{attribute 'linkalways'} 
{attribute 'no_explicit_call' := 'This FB is a CLASS and must be accessed using methods or properties'}
{attribute 'enable_dynamic_creation'}
FUNCTION_BLOCK Node_F_VN_AppendToContainer_ITcVnContainer EXTENDS VisionNode
VAR
    ipElement : _ITcVnContainer;
    ipContainer : _ITcVnContainer;
    hrPrev : _HRESULT(S_OK);
	hresult : _HRESULT(S_OK);
END_VAR

METHOD PUBLIC  Clone : I_Node
VAR
	pNode : POINTER TO Node_F_VN_AppendToContainer_ITcVnContainer;
END_VAR
pNode := __NEW(Node_F_VN_AppendToContainer_ITcVnContainer);
Clone := pNode^;
END_METHOD

METHOD FB_init : BOOL
VAR_INPUT
	bInitRetains : BOOL; // if TRUE, the retain variables are initialized (warm start / cold start)
	bInCopyCode : BOOL;  // if TRUE, the instance afterwards gets moved into the copy code (online change)
END_VAR
AddInput('ipElement', ipElement);
AddInput('ipContainer', ipContainer);
AddInput('hrPrev', hrPrev);
AddOutput('ipContainer', ipContainer);
AddOutput('hresult',hresult);
END_METHOD

METHOD PROTECTED OnExecute : HRESULT
hresult.Value := F_VN_AppendToContainer_ITcVnContainer(
    ipElement := ipElement.Value,
	ipContainer := ipContainer.Value,
	hrPrev:= hrPrev.Value);
END_METHOD

METHOD PUBLIC PreExecutionCheck
VAR_INPUT
	Check : I_PreExecutionChecks;
END_VAR
Check.IsTrue(ipContainer.IsValid, 'ipContainer must be a valid container');
END_METHOD

END_FUNCTION_BLOCK

(* stored: Version 1.1.0.1, ProductVersion 3.1.4024.13
   POU Node_F_VN_AppendToContainer_ITcVnContainer: Id {16faa72d-9e4b-4692-b20a-b0f3b6fa5e87}, SpecialFunc None
   Folder Constructor: Id {ae4da694-88f2-47ef-8374-be6125b8ea3d}
   Method Clone: Id {c03d167a-5f53-48c3-88bb-1a3c34f9a65d}
   Method FB_init: Id {1caf2c53-8deb-414f-8e3e-db88aa8762d7}
   Method OnExecute: Id {2717e6aa-8ffd-4f75-9c1a-704121a9e3f9}
   Method PreExecutionCheck: Id {254e989a-e7d1-409c-9da0-c05029184d0f} *)
